PROGRAM PRG_TestComponents
VAR
	// Interfaces
	iComponent1, iComponet2, iComponet3 : I_TestComponent;	

	// Componentes
	Component_1 : FB_Test_Component := (Name := 'TC-01');
	Component_2 : FB_Test_Component := (Name := 'TC-02');
	Component_3 : FB_Test_Component := (Name := 'TC-03');

	// Test Triggers
	Trig1a, Trig1b, Trig2a, Trig2b, Trig3a, Trig3b : BOOL;
END_VAR

M_Map();

METHOD M_Map : BOOL
VAR_INPUT
END_VAR
// Map Interface
iComponent1 := Component_1;
iComponet2 := Component_2;
iComponet3 := Component_3;

// Map Parameters
Component_1.pTrig := Trig1a;
Component_1.pTrig2 := Trig1b;
Component_2.pTrig := Trig2a;
Component_2.pTrig2 := Trig2b;
Component_3.pTrig := Trig3a;
Component_3.pTrig2 := Trig3b;

// Cylic Calls
Component_1.M_CyclicLogic();
Component_2.M_CyclicLogic();
Component_3.M_CyclicLogic();
END_METHOD

END_PROGRAM

(* stored: Version 1.1.0.1
   POU PRG_TestComponents: Id {31b2772e-2b0b-45e6-a2be-c8f1d02a4d59}, SpecialFunc None
   Method M_Map: Id {feb471fa-b931-4c00-80f4-b70de2e8d9bd} *)
